FUNCTION Camera_Get_Int : Buffer_Error
VAR_INPUT
	Camera : REFERENCE TO Cognex_Camera;
	Num : USINT;
END_VAR

VAR_IN_OUT
	Out : INT;
END_VAR

Camera_Get_Int := Get_Int_From_Buffer(	Num:= Num, 
										Layout:= Camera.Input_Buffer_Layout, 
										Buffer:= Camera.User_Data.Data, 
										Out:= Out);

END_FUNCTION

(* stored: Version 1.1.0.1, ProductVersion 3.1.4024.10
   POU Camera_Get_Int: Id {b74ad591-15d3-4de3-a6b8-2c74aa6d2bf6}, SpecialFunc None *)
